FUNCTION_BLOCK Q_ChildPosition (* Command change child position ( Part 6 - F.16 ) *)
  (* Standard: ISO 11783-6; Description: Copyright (c) 2022 HR Agrartechnik GmbH This program and the accompanying materials are made available under the terms of the Eclipse Public License 2.0 which is available at https://www.eclipse.org/legal/epl-2.0/ SPDX-License-Identifier: EPL-2.0 see Description Tab *)
  (* Version 1.0, 2022-07-08, Franz Höpfinger, HR Agrartechnik GmbH *)
  PACKAGE isobus::UT::Q;
  IMPORT isobus::UT::Q::const::IDs::ID_NULL;
  (* Documentation:
  Command change child position ( Part 6 - F.16 )
   The Change Child Position command is used to change the absolute position of an object.
   Valid Object IDs
   A child position Object ID is valid if it falls within one of the following ISO 11783-6 ID ranges:
    - Container: 3000 – 3999
   - Button: 6000 – 6999
   - InputBooleanField: 7000 – 7999
   - InputStringField: 8000 – 8999
   - InputNumberField: 9000 – 9999
   - InputListField: 10000 – 10999
   - OutputStringField: 11000 – 11999
   - OutputNumberField: 12000 – 12999
   - TypLine: 13000 – 13999
   - TypRectangle: 14000 – 14999
   - TypEllipse: 15000 – 15999
   - TypPolygon: 16000 – 16999
   - Meter: 17000 – 17999
   - LinearBarGraph: 18000 – 18999
   - ArchedBarGraph: 19000 – 19999
   - PictureGraphic: 20000 – 20499
   - ObjectPointer: 27000 – 27999
   - OutputListObject: 37000 – 37999
   - ExternalObjectPointer: 43000 – 43999
   - AnimationObject: 44000 – 44999
   - ScaledGraphicObject: 48000 – 48999
   - AuxiliaryFunction: 29000 – 29999
   - AuxiliaryFunctionType2: 31000 – 31999
   - AuxiliaryInput: 30000 – 30999
   - AuxiliaryInputType2: 32000 – 32999
   - AuxiliaryControlDesignator: 33000 – 33999
    ID_NULL (65535) is not a command target but can be used in INIT to deactivate the FB. Any ID outside these ranges is invalid for commanding.
   Activate / Deactivate
   The FB is deactivated by default. It becomes active when INIT provides a valid child position Object ID. Sending INIT with ID_NULL (65535) deactivates the FB again. This toggle can be repeated arbitrarily.
    - INIT + ID_NULL (65535): FB deactivated, STATUS="DEACTIVATED", s16result=VT_E_DEACTIVATED (-40)
   - INIT + valid child position ID: FB activated, STATUS="initialized", s16result=VT_E_NO_ERR (0). If a REQ was buffered before, it is executed immediately.
   - INIT + invalid ID: STATUS="ERROR: Invalid Object ID (not a child position object)", s16result=VT_E_INVALID_OBJECT_ID (-132)
    REQ Handling
    - REQ before any INIT: Buffered, STATUS="Buffered: INIT not yet completed", s16result=VT_E_NOT_READY (-131)
   - REQ while deactivated (INIT came with NULL or invalid ID): STATUS shows the actual deactivation reason, s16result=VT_E_DEACTIVATED (-40) or VT_E_INVALID_OBJECT_ID (-132)
   - REQ while active: Command sent to VT, result reflected in CNF
    param[in] {objectID, uint16_t}
   Object ID. Use ID_NULL (65535) to deactivate the FB. Use a valid child position object ID to activate.
   param[in] {parentObjectID, uint16_t}
   Parent object ID
   param[in] {xPosition, uint16_t}
   New X position relative to the top left corner of parent object
   param[in] {yPosition, uint16_t}
   New Y position relative to the top left corner of parent object.
   Return Values (s16result):
   int16_t
    - VT_E_NO_ERR (0) - OK
   - VT_E_DEACTIVATED (-40) - FB deactivated (INIT received with ID_NULL)
   - VT_E_INVALID_OBJECT_ID (-132) - Object ID is invalid (not a child position object)
   - VT_E_NOT_READY (-131) - Buffered: INIT not yet completed
   - VT_E_OVERFLOW (-6) - buffer overflow
   - VT_E_NOACT (-8) - Command not possible in current state
   - VT_E_NO_INSTANCE (-21) - No VT client available
   - VT_E_ISO_INSTANCE_INVALID (-129) - Identifier for instance (connection) invalid
   - VT_E_NOT_ALIVE (-130) - Identifier for instance valid, but VT Dead.
  *)
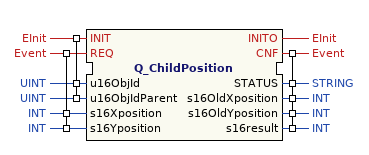
  EVENT_INPUT
    INIT : EInit WITH u16ObjId, u16ObjIdParent; (* Service Initialization *)
    REQ WITH s16Xposition, s16Yposition; (* Service Request *)
  END_EVENT
  EVENT_OUTPUT
    INITO : EInit; (* Initialization Confirm *)
    CNF WITH STATUS, s16OldYposition, s16OldXposition, s16result; (* Confirmation of Requested Service *)
  END_EVENT
  VAR_INPUT
    u16ObjId : UINT := ID_NULL; (* Object ID *)
    u16ObjIdParent : UINT := ID_NULL; (* Parent object ID *)
    s16Xposition : INT; (* New X position relative to the top left corner of parent object *)
    s16Yposition : INT; (* New Y position relative to the top left corner of parent object *)
  END_VAR
  VAR_OUTPUT
    STATUS : STRING; (* Service Status *)
    s16OldXposition : INT; (* Old X position relative to the top left corner of parent object *)
    s16OldYposition : INT; (* Old Y position relative to the top left corner of parent object *)
    s16result : INT; (* retval see description *)
  END_VAR
END_FUNCTION_BLOCK
